% RSLogix 500 project ONE BUTTON LATCH-UNLATCH_BAK007.RSS, saved by version 10.00.00.00 %
PROJECT "UNTITLED"    % processor: Bul.1763 MicroLogix 1100 Series B %

PROGRAM FILES
  LAD 2   4 rungs

DATA FILES
  O0 OUTPUT  4 elements
  I1 INPUT  6 elements
  S2 STATUS  66 elements
  B3 BINARY  2 elements
  T4 TIMER  1 elements
  C5 COUNTER  1 elements
  R6 CONTROL  1 elements
  N7 INTEGER  1 elements
  F8 FLOAT  1 elements

LADDER 2
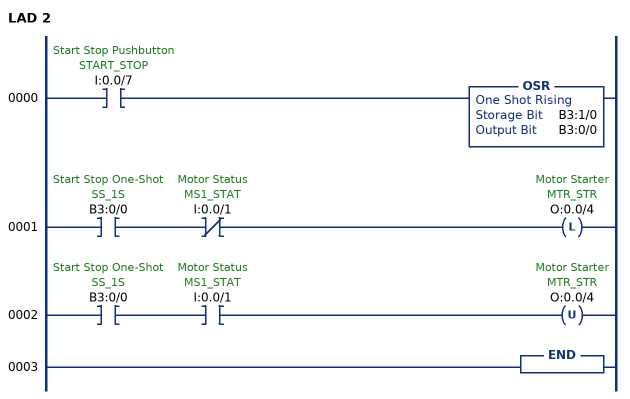
% Rung: 0 %
SOR XIC I:0.0/7 OSR B3:1/0 B3:0/0 EOR
%   I:0.0/7  START_STOP  "Start Stop Pushbutton" %
%   B3:0/0  SS_1S  "Start Stop One-Shot" %
% Rung: 1 %
SOR XIC B3:0/0 XIO I:0.0/1 OTL O:0.0/4 EOR
%   B3:0/0  SS_1S  "Start Stop One-Shot" %
%   I:0.0/1  MS1_STAT  "Motor Status" %
%   O:0.0/4  MTR_STR  "Motor Starter" %
% Rung: 2 %
SOR XIC B3:0/0 XIC I:0.0/1 OTU O:0.0/4 EOR
%   B3:0/0  SS_1S  "Start Stop One-Shot" %
%   I:0.0/1  MS1_STAT  "Motor Status" %
%   O:0.0/4  MTR_STR  "Motor Starter" %
% Rung: 3 %
SOR END EOR

OTHER DOCUMENTED ADDRESSES
  B3:0/1  RED_OS  "Red One-Shot"
  O:0.0/0  GRN_LT  "Green Light"
  O:0.0/2  RED_LT  "Red Light"
